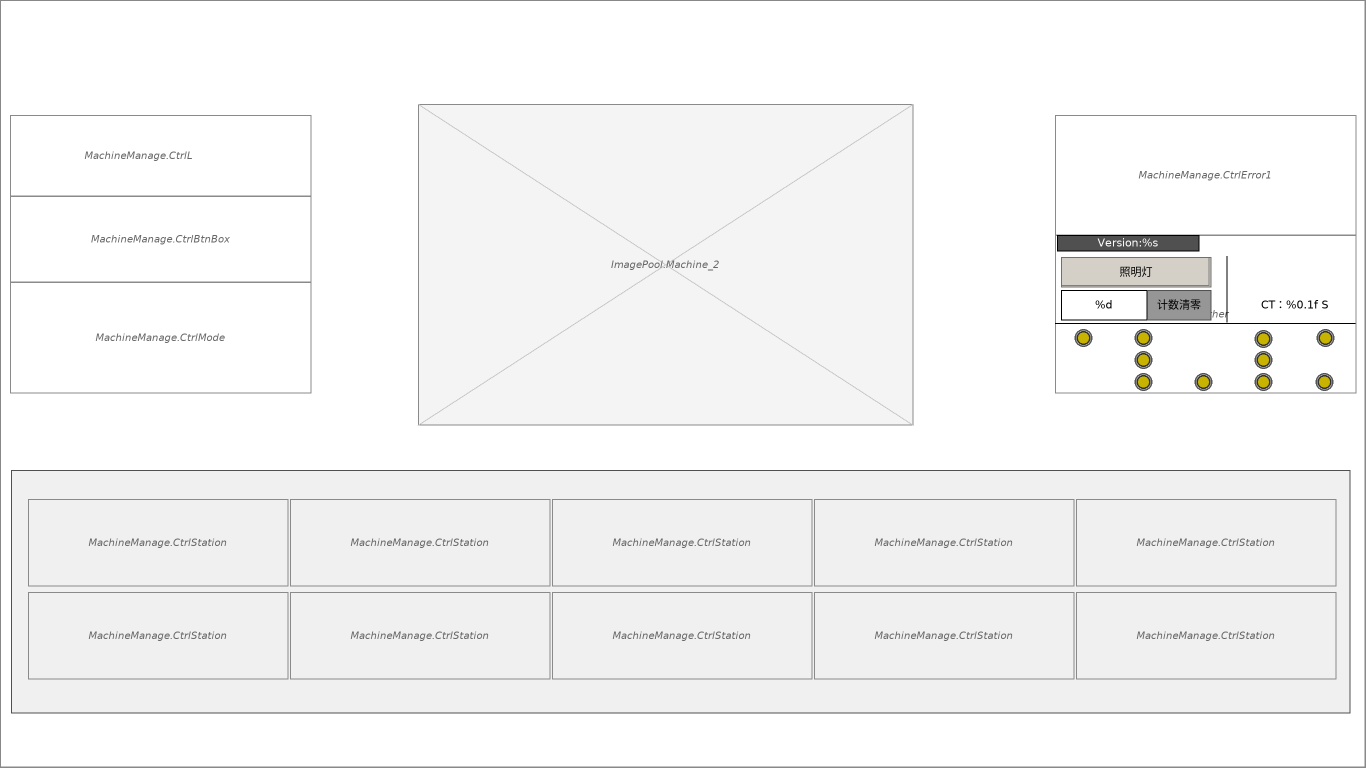
VISUALIZATION PageHome  // 1366x768
    Frame (0,0 1366x768)
        shows FrameMain()
    Frame (10,115 301x81)
        shows MachineManage.CtrlLanguage(System := G_stSystem)
    Frame (10,196 301x86)
        shows MachineManage.CtrlBtnBox(System := G_stSystem)
    Frame (10,282 301x111)
        shows MachineManage.CtrlMode(System := G_stSystem)
    Frame (1055,115 301x120)
        shows MachineManage.CtrlError1(System := G_stSystem, Error := G_stError.stNow)
    Frame (1055,235 301x158), text variable: P_System._fbCT.CycleTime
        shows CtrlOther()
    Rectangle (192,135 83x56)
    Button (1061,257 150x30), "照明灯"
        toggle GVL.Q.bLED
    Line (1227,322) (1227,256)
    Image (418,104 495x321), image: ImagePool.Machine_2
    Rectangle (1242,257 106x30), text list: 'MachineType', text index: GVL_Data.stRecipe.eMachineType
    Rectangle (1057,235 142x16), "Version:%s", text variable: MAIN.VERSION
    Rectangle (1242,290 106x30), "CT：%0.1f S", text variable: P_System._cttime
    Rectangle (1061,290 86x30), "%d", text variable: P_System._iProductionCount
    Rectangle (1147,290 64x30), "计数清零"
        tap P_System._bCountZero
    Lamp1 (1072,328 23x20), variable: GVL.I.bLine0Check2, style: Lamp-Lamp1-Yellow
    Line (1055,323) (1355,323)
    Lamp1 (1132,372 23x20), variable: GVL.I.bSteeringCheck1, style: Lamp-Lamp1-Yellow
    Lamp1 (1132,328 23x20), variable: GVL.I.bLine0Check3, style: Lamp-Lamp1-Yellow
    Lamp1 (1252,329 23x20), variable: GVL.I.bUnloadUcCheck2, style: Lamp-Lamp1-Yellow
    Lamp1 (1314,328 23x20), variable: GVL.I.bUnloadFrockConveyorCheck2, style: Lamp-Lamp1-Yellow
    Lamp1 (1192,372 23x20), variable: GVL.I.bOpenLockCheck, style: Lamp-Lamp1-Yellow
    Lamp1 (1252,372 23x20), variable: GVL.I.bTakeUcCheck1, style: Lamp-Lamp1-Yellow
    Lamp1 (1313,372 23x20), variable: GVL.I.bUnloadFrockCheck1, style: Lamp-Lamp1-Yellow
    Lamp1 (1132,350 23x20), variable: GVL.I.bAcquireCheck2, style: Lamp-Lamp1-Yellow
    Lamp1 (1252,350 23x20), variable: GVL.I.bUnloadUcCheck1, style: Lamp-Lamp1-Yellow
    Rectangle (11,470 1339x243)
    Frame (290,592 260x87)
        shows MachineManage.CtrlStation(System := G_stSystem, Station := G_arrStation[5])
    Frame (552,592 260x87)
        shows MachineManage.CtrlStation(System := G_stSystem, Station := G_arrStation[6])
    Frame (814,592 260x87)
        shows MachineManage.CtrlStation(System := G_stSystem, Station := G_arrStation[7])
    Frame (1076,592 260x87)
        shows MachineManage.CtrlStation(System := G_stSystem, Station := G_arrStation[8])
    Frame (1076,499 260x87)
        shows MachineManage.CtrlStation(System := G_stSystem, Station := G_arrStation[9])
    Frame (28,499 260x87)
        shows MachineManage.CtrlStation(System := G_stSystem, Station := G_arrStation[0])
    Frame (290,499 260x87)
        shows MachineManage.CtrlStation(System := G_stSystem, Station := G_arrStation[1])
    Frame (552,499 260x87)
        shows MachineManage.CtrlStation(System := G_stSystem, Station := G_arrStation[2])
    Frame (814,499 260x87)
        shows MachineManage.CtrlStation(System := G_stSystem, Station := G_arrStation[3])
    Frame (28,592 260x87)
        shows MachineManage.CtrlStation(System := G_stSystem, Station := G_arrStation[4])
END_VISUALIZATION

(* stored: Version 1.1.0.1, ProductVersion 3.1.4024.3
   Visu PageHome: Id {6f3cc229-475a-49a0-905f-190a42f85a9f} *)
